FUNCTION_BLOCK UNIT_Observer (* Owns all cell sensors (shared by several skills): periodic sampling through IO primitives, state observer, published state variables (AID/Operational data) *)
  (* Standard: 61499-2 *)
  (* Version 2.0, 2026-09-27, Project contributors, Filling cell reference model *)
  PACKAGE fillingcell;
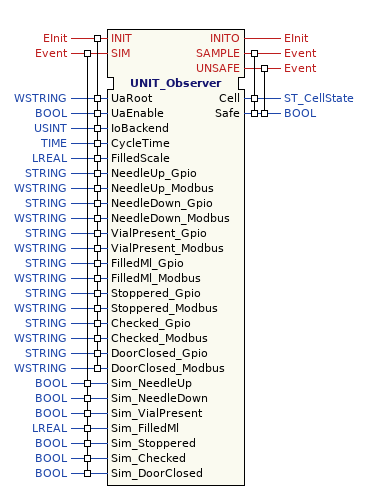
  EVENT_INPUT
    INIT : EInit WITH UaRoot, UaEnable, IoBackend, CycleTime, FilledScale, NeedleUp_Gpio, NeedleUp_Modbus, NeedleDown_Gpio, NeedleDown_Modbus, VialPresent_Gpio, VialPresent_Modbus, FilledMl_Gpio, FilledMl_Modbus, Stoppered_Gpio, Stoppered_Modbus, Checked_Gpio, Checked_Modbus, DoorClosed_Gpio, DoorClosed_Modbus;
    SIM WITH Sim_NeedleUp, Sim_NeedleDown, Sim_VialPresent, Sim_FilledMl, Sim_Stoppered, Sim_Checked, Sim_DoorClosed;
  END_EVENT
  EVENT_OUTPUT
    INITO : EInit;
    SAMPLE WITH Cell, Safe;
    UNSAFE WITH Safe;
  END_EVENT
  VAR_INPUT
    UaRoot : WSTRING;
    UaEnable : BOOL;
    IoBackend : USINT;
    CycleTime : TIME := T#100ms;
    FilledScale : LREAL := 0.01;
    NeedleUp_Gpio : STRING;
    NeedleUp_Modbus : WSTRING;
    NeedleDown_Gpio : STRING;
    NeedleDown_Modbus : WSTRING;
    VialPresent_Gpio : STRING;
    VialPresent_Modbus : WSTRING;
    FilledMl_Gpio : STRING;
    FilledMl_Modbus : WSTRING;
    Stoppered_Gpio : STRING;
    Stoppered_Modbus : WSTRING;
    Checked_Gpio : STRING;
    Checked_Modbus : WSTRING;
    DoorClosed_Gpio : STRING;
    DoorClosed_Modbus : WSTRING;
    Sim_NeedleUp : BOOL;
    Sim_NeedleDown : BOOL;
    Sim_VialPresent : BOOL;
    Sim_FilledMl : LREAL;
    Sim_Stoppered : BOOL;
    Sim_Checked : BOOL;
    Sim_DoorClosed : BOOL;
  END_VAR
  VAR_OUTPUT
    Cell : fillingcell::ST_CellState;
    Safe : BOOL;
  END_VAR
  FBS
    Ids : fillingcell::UA_ObserverIds;
    In_NeedleUp : fillingcell::IO_DI;
    In_NeedleDown : fillingcell::IO_DI;
    In_VialPresent : fillingcell::IO_DI;
    In_FilledMl : fillingcell::IO_AI;
    In_Stoppered : fillingcell::IO_DI;
    In_Checked : fillingcell::IO_DI;
    In_DoorClosed : fillingcell::IO_DI;
    Publisher : iec61499::net::PUBLISH_9;
    Obs : fillingcell::FC_Observer;
    Cycle : iec61499::events::E_CYCLE;
  END_FBS
  EVENT_CONNECTIONS
    INIT TO Ids.INIT;
    Ids.INITO TO In_NeedleUp.INIT;
    In_NeedleUp.INITO TO In_NeedleDown.INIT;
    In_NeedleDown.INITO TO In_VialPresent.INIT;
    In_VialPresent.INITO TO In_FilledMl.INIT;
    In_FilledMl.INITO TO In_Stoppered.INIT;
    In_Stoppered.INITO TO In_Checked.INIT;
    In_Checked.INITO TO In_DoorClosed.INIT;
    In_DoorClosed.INITO TO Publisher.INIT;
    Publisher.INITO TO INITO;
    Publisher.INITO TO Cycle.START;
    Cycle.EO TO In_NeedleUp.REQ;
    In_NeedleUp.CNF TO In_NeedleDown.REQ;
    In_NeedleDown.CNF TO In_VialPresent.REQ;
    In_VialPresent.CNF TO In_FilledMl.REQ;
    In_FilledMl.CNF TO In_Stoppered.REQ;
    In_Stoppered.CNF TO In_Checked.REQ;
    In_Checked.CNF TO In_DoorClosed.REQ;
    In_DoorClosed.CNF TO Obs.SAMPLE;
    Obs.CNF TO SAMPLE;
    Obs.CNF TO Publisher.REQ;
    Obs.UNSAFE TO UNSAFE;
  END_CONNECTIONS
  DATA_CONNECTIONS
    IoBackend TO In_NeedleUp.Backend;
    NeedleUp_Gpio TO In_NeedleUp.GpioName;
    NeedleUp_Modbus TO In_NeedleUp.ModbusId;
    Sim_NeedleUp TO In_NeedleUp.SimValue;
    IoBackend TO In_NeedleDown.Backend;
    NeedleDown_Gpio TO In_NeedleDown.GpioName;
    NeedleDown_Modbus TO In_NeedleDown.ModbusId;
    Sim_NeedleDown TO In_NeedleDown.SimValue;
    IoBackend TO In_VialPresent.Backend;
    VialPresent_Gpio TO In_VialPresent.GpioName;
    VialPresent_Modbus TO In_VialPresent.ModbusId;
    Sim_VialPresent TO In_VialPresent.SimValue;
    IoBackend TO In_FilledMl.Backend;
    FilledMl_Gpio TO In_FilledMl.GpioName;
    FilledMl_Modbus TO In_FilledMl.ModbusId;
    Sim_FilledMl TO In_FilledMl.SimValue;
    FilledScale TO In_FilledMl.Scale;
    IoBackend TO In_Stoppered.Backend;
    Stoppered_Gpio TO In_Stoppered.GpioName;
    Stoppered_Modbus TO In_Stoppered.ModbusId;
    Sim_Stoppered TO In_Stoppered.SimValue;
    IoBackend TO In_Checked.Backend;
    Checked_Gpio TO In_Checked.GpioName;
    Checked_Modbus TO In_Checked.ModbusId;
    Sim_Checked TO In_Checked.SimValue;
    IoBackend TO In_DoorClosed.Backend;
    DoorClosed_Gpio TO In_DoorClosed.GpioName;
    DoorClosed_Modbus TO In_DoorClosed.ModbusId;
    Sim_DoorClosed TO In_DoorClosed.SimValue;
    UaRoot TO Ids.UaRoot;
    UaEnable TO Publisher.QI;
    Ids.IdPub TO Publisher.ID;
    CycleTime TO Cycle.DT;
    In_NeedleUp.IN TO Obs.NeedleUp;
    In_NeedleDown.IN TO Obs.NeedleDown;
    In_VialPresent.IN TO Obs.VialPresent;
    In_FilledMl.IN TO Obs.FilledMl;
    In_Stoppered.IN TO Obs.Stoppered;
    In_Checked.IN TO Obs.Checked;
    In_DoorClosed.IN TO Obs.DoorClosed;
    Obs.Cell TO Cell;
    Obs.Safe TO Safe;
    Obs.O_NeedleUp TO Publisher.SD_1;
    Obs.O_NeedleDown TO Publisher.SD_2;
    Obs.O_VialPresent TO Publisher.SD_3;
    Obs.O_FilledMl TO Publisher.SD_4;
    Obs.O_Stoppered TO Publisher.SD_5;
    Obs.O_Checked TO Publisher.SD_6;
    Obs.O_DoorClosed TO Publisher.SD_7;
    Obs.O_Valid TO Publisher.SD_8;
    Obs.O_Safe TO Publisher.SD_9;
  END_CONNECTIONS
END_FUNCTION_BLOCK
